TYPE TcaTwinSAFEConfig :
STRUCT
END_STRUCT
END_TYPE

(* stored: Version 1.1.0.1
   DUT TcaTwinSAFEConfig: Id {fd052477-d444-4584-a6e7-a2945850364e} *)
